FUNCTION_BLOCK CLIENT_2_1 (* 2 SD/1 RD Client Interface *)
  (* Standard: 61499-1; Function: Communication; Description: 2SD/1RD Client *)
  (* Version 0.1, 2006-04-26, JHC, Holobloc Inc, Added service sequences. *)
  (* Version 0.0, 2000-12-31, JHC, Rockwell Automation *)
  (* Compiler header: package fb.rt.net; *)
  (* Compiler Java Sun JDK 1.5.0 *)
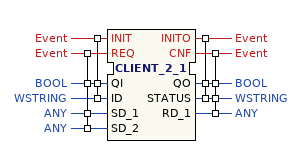
  EVENT_INPUT
    INIT WITH QI, ID; (* Service Initialization *)
    REQ WITH QI, SD_1, SD_2; (* Service Request *)
  END_EVENT
  EVENT_OUTPUT
    INITO WITH QO, STATUS; (* Initialization Confirm *)
    CNF WITH QO, STATUS, RD_1; (* Service Confirmation *)
  END_EVENT
  VAR_INPUT
    QI : BOOL; (* Event Input Qualifier *)
    ID : WSTRING; (* Connection Identifier *)
    SD_1 : ANY; (* Data to Send *)
    SD_2 : ANY; (* Data to Send *)
  END_VAR
  VAR_OUTPUT
    QO : BOOL; (* Event Output Qualifier *)
    STATUS : WSTRING; (* Service Status *)
    RD_1 : ANY; (* Received Data *)
  END_VAR
  SERVICE CLIENT/SERVER
    SEQUENCE normal_establishment
      SERVER.INIT+(ID) -> SERVER.INITO+();
      CLIENT.INIT+(ID) -> SERVER.connect(ID) -> CLIENT.INITO+();
    END_SEQUENCE
    SEQUENCE bad_server_ID
      SERVER.INIT+(ID) -> SERVER.INITO-(STATUS);
    END_SEQUENCE
    SEQUENCE bad_client_ID
      CLIENT.INIT+(ID) -> CLIENT.INITO-(STATUS);
    END_SEQUENCE
    SEQUENCE connection_refused
      CLIENT.INIT+(ID) -> SERVER.connect() -> CLIENT.INITO-(STATUS);
    END_SEQUENCE
    SEQUENCE normal_data_transfer
      CLIENT.REQ+(SD_1,SD_2) -> SERVER.IND+(RD_1,RD_2);
      SERVER.RSP+(SD_1) -> CLIENT.CNF+(RD_1);
    END_SEQUENCE
    SEQUENCE request_inhibited
      CLIENT.REQ-() -> CLIENT.CNF-(STATUS);
    END_SEQUENCE
    SEQUENCE server_decode_error (* Causes disconnection *)
      CLIENT.REQ+(SD) -> SERVER.decode(RD_1,RD_2) -> CLIENT.INITO-(STATUS) -> SERVER.INITO-(STATUS);
    END_SEQUENCE
    SEQUENCE client_decode_error (* Causes disconnection *)
      SERVER.CNF+(SD_1) -> CLIENT.decode(RD_1) -> SERVER.INITO-(STATUS) -> CLIENT.INITO-(STATUS);
    END_SEQUENCE
    SEQUENCE client_initiated_termination
      CLIENT.INIT-() -> SERVER.INITO-(STATUS) -> CLIENT.INITO-(STATUS);
    END_SEQUENCE
    SEQUENCE server_initiated_termination
      SERVER.INIT-() -> CLIENT.INITO-(STATUS) -> SERVER.INITO-(STATUS);
    END_SEQUENCE
    SEQUENCE system_initiated_termination
      -> CLIENT.INITO-(STATUS);
      -> SERVER.INITO-(STATUS);
    END_SEQUENCE
  END_SERVICE
END_FUNCTION_BLOCK
